TYPE aocHmiStatus_TypeStruct :
STRUCT
	
	automaticOrderChangeStatus	: STRING;

END_STRUCT
END_TYPE

(* stored: Version 1.1.0.1
   DUT aocHmiStatus_TypeStruct: Id {faf56f49-1438-4c27-ae08-6040110fb1b1} *)
